// TIA Portal V20 export
// export: Created 2025-12-01T14:57:23.1457372Z, ExportSetting None, DisplayName Totally Integrated Automation Portal, DisplayVersion V20 Update 3, DisplayName TIA Portal Openness, DisplayVersion V20 Update 3, DisplayName TIA Portal Version Control Interface, DisplayVersion V20 Update 3, DisplayName STEP 7 Professional, DisplayVersion V20 Update 3, DisplayName STEP 7 Safety, DisplayVersion V20 Update 2, DisplayName WinCC Basic/Comfort/Advanced, DisplayVersion V20 Update 3, DisplayName WinCC Professional, DisplayVersion V20 Update 3, DisplayName WinCC Unified, DisplayVersion V20 Update 3
DATA_BLOCK "DB912_Tipo_Scanner_Router"   // DB912
{ S7_Optimized_Access := 'FALSE' }
AUTHOR : ROUTER
NAME : 20170522
VERSION : 3.2
// El 20170522 se incluyen las modificaciones para poder recibir y tratar mensajes INIR para varios bucles.
// stored: AutoNumber false
   VAR RETAIN
      SCANNER { S7_SetPoint := 'True'} : Array[0.."ROUT_Max_Scanners"] of "ROUT_Def_Scanner";
   END_VAR
BEGIN
   SCANNER[1..8].Tipo := 1;
   SCANNER[1].Bit_Ini_Ordenes := 1;
   SCANNER[2].Bit_Ini_Ordenes := 2;
   SCANNER[3].Bit_Ini_Ordenes := 3;
   SCANNER[4].Bit_Ini_Ordenes := 4;
   SCANNER[5].Bit_Ini_Ordenes := 5;
   SCANNER[6].Bit_Ini_Ordenes := 6;
   SCANNER[7].Bit_Ini_Ordenes := 7;
   SCANNER[8].Bit_Ini_Ordenes := 8;
   SCANNER[12].Bit_Ini_Ordenes := 7;
   SCANNER[21].Bit_Ini_Ordenes := 10;
   SCANNER[22].Bit_Ini_Ordenes := 11;
   SCANNER[23].Bit_Ini_Ordenes := 12;
   SCANNER[24].Bit_Ini_Ordenes := 13;
   SCANNER[25].Bit_Ini_Ordenes := 14;
   SCANNER[26].Bit_Ini_Ordenes := 15;
   SCANNER[27].Bit_Ini_Ordenes := 16;
   SCANNER[28].Bit_Ini_Ordenes := 17;
   SCANNER[29].Bit_Ini_Ordenes := 18;
   SCANNER[30].Bit_Ini_Ordenes := 19;
   SCANNER[31].Bit_Ini_Ordenes := 20;
   SCANNER[32].Bit_Ini_Ordenes := 21;
   SCANNER[114].Bit_Ini_Ordenes := 3;
   SCANNER[115].Bit_Ini_Ordenes := 2;
   SCANNER[116].Bit_Ini_Ordenes := 1;
   SCANNER[2..8].N_Bits_Orden := 1;
   SCANNER[1].Num_Inicializacion := -1;
   SCANNER[2].Num_Inicializacion := 2;
   SCANNER[3].Num_Inicializacion := 3;
   SCANNER[4].Num_Inicializacion := 4;
   SCANNER[5].Num_Inicializacion := 5;
   SCANNER[6].Num_Inicializacion := 6;
   SCANNER[7].Num_Inicializacion := 7;
   SCANNER[8].Num_Inicializacion := 8;
END_DATA_BLOCK
